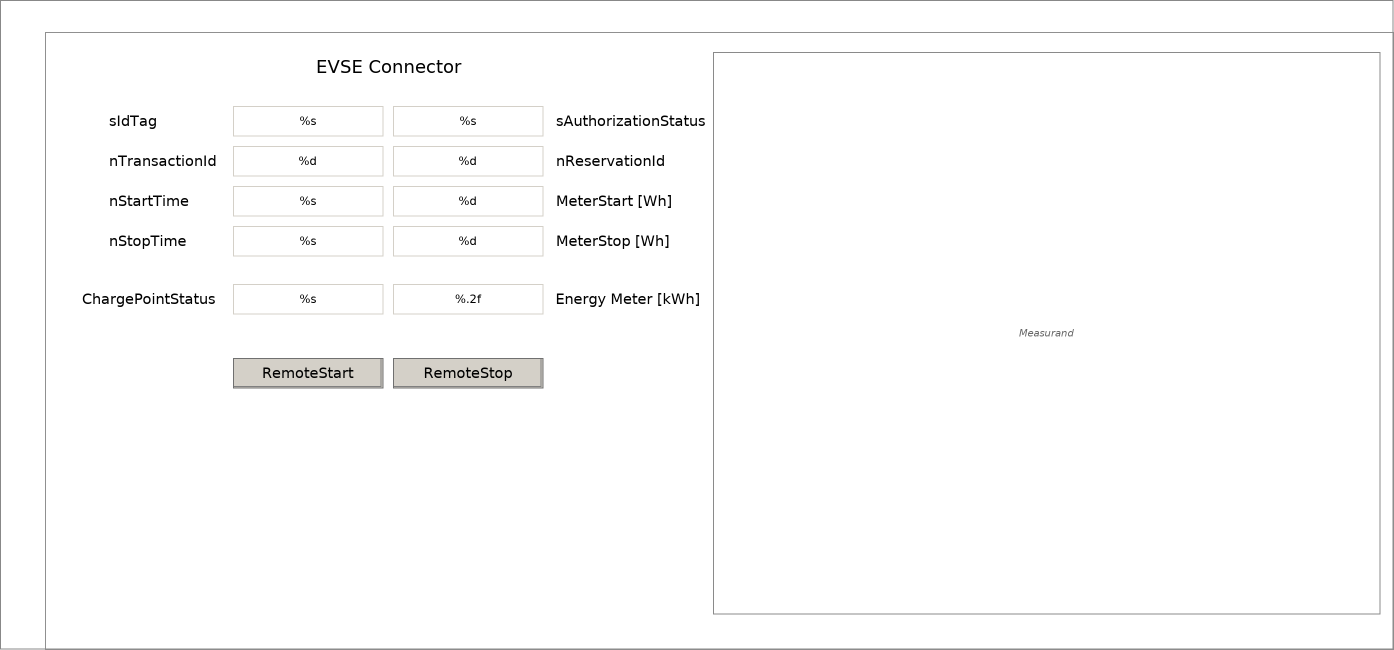
VISUALIZATION Visu_Connector  // 1394x650
VAR_IN_OUT
	stConnector : ST_Connector; 
 	fbMeasurand : FB_SampledValueMeasurands; 
	bRemoteStart : BOOL;
	bRemoteStop : BOOL; 
END_VAR
    GroupBox (45,24 1349x626)
        Textfield (188,82 150x30), "%s", text variable: stConnector.sIdTag
        Label (61,82 117x30), "sIdTag"
        Textfield (188,122 150x30), "%d", text variable: stConnector.nTransactionID
        Textfield (188,162 150x30), "%s", text variable: stConnector.sStartTime
        Textfield (188,202 150x30), "%s", text variable: stConnector.sStopTime
        Label (61,122 117x30), "nTransactionId"
        Label (61,162 117x30), "nStartTime"
        Label (61,202 117x30), "nStopTime"
        Textfield (348,82 150x30), "%s", text variable: stConnector.sAuthorizationStatus
        Textfield (188,260 150x30), "%s", text variable: stConnector.sChargpointStatus
        Label (29,260 150x30), "ChargePointStatus"
        Textfield (348,162 150x30), "%d", text variable: stConnector.nMeterStart
        Label (508,162 150x30), "MeterStart [Wh]"
        Textfield (348,202 150x30), "%d", text variable: stConnector.nMeterStop
        Label (508,202 150x30), "MeterStop [Wh]"
        Label (508,82 150x30), "sAuthorizationStatus"
        Textfield (348,122 150x30), "%d", text variable: stConnector.nReservationId
        Label (508,122 150x30), "nReservationId"
        Textfield (348,260 150x30), "%.2f", text variable: fbMeasurand.fEnergyActiveImportRegister
        Label (508,260 150x30), "Energy Meter [kWh]"
        Label (261,28 166x30), "EVSE Connector"
        Button (188,334 150x30), "RemoteStart"
            tap bRemoteStart
        Button (348,334 150x30), "RemoteStop"
            tap bRemoteStop
        Frame (668,28 667x562)
            shows Measurand(fbMeasurand := fbMeasurand)
END_VISUALIZATION

(* stored: Version 1.1.0.1
   Visu Visu_Connector: Id {3154e44a-2d9d-4fe5-b245-1993b01c69a7} *)
